Fanuc KAREL source: kt00405.KL

-- PROVISIONAL review KL for V1013-1; original PC SHA256 d02ce8dd29aeec4519ce106d0438d064a054909856b1c59b98b6211a64b51add
-- Incomplete behavior may be omitted. Consult companion uncertainty JSON. Do not deploy.
PROGRAM KT00405
%NOLOCKGROUP
VAR
  R1 : REAL
  I2 : INTEGER
  OUT : BOOLEAN
BEGIN
  -- UNRESOLVED_PC offsets 5-16; opcodes 2E,23
  -- UNRESOLVED_PC offsets 21-32; opcodes 2E,23
  -- UNRESOLVED_PC offsets 37-57; opcodes 21,21,64,71,23
  -- UNRESOLVED_PC offsets 62-66; opcodes 7F
END KT00405
